// TwinCAT 3 PLC project PI_test
// ProgramVersion: 3.1.4024.0
// libraries:
//   Tc2_ControllerToolbox, * (Beckhoff Automation GmbH)
//   Tc2_Standard, * (Beckhoff Automation GmbH)
//   Tc2_System, * (Beckhoff Automation GmbH)
//   Tc3_Module, * (Beckhoff Automation GmbH)
// project tree:
//   / PlcTask.TcTTO
//   POUs/ FB_FILL_SIM.TcPOU, TYP_VESSEL.TcDUT, MAIN.TcPOU
// real-time tasks:
//   TASK PlcTask: cycle T#1ms, priority 20, ADS port 350

CONFIGURATION PI_test
    RESOURCE PLC ON TwinCAT3
        TASK PlcTask(INTERVAL := T#1ms, PRIORITY := 20);
        PROGRAM MAIN WITH PlcTask : MAIN;
    END_RESOURCE
END_CONFIGURATION

// ---- POUs/TYP_VESSEL.TcDUT
TYPE TYP_VESSEL :
STRUCT
	rVesselSize: LREAL := 100;
	rFillingRate: LREAL := 100;
	rValveInOpening: LREAL := 50;
	rEmptyingRate: LREAL := 100;
	rValveOutOpening: LREAL := 50;
	rSetPoint: LREAL := 50;
	bReset: BOOL;
END_STRUCT
END_TYPE

// ---- POUs/MAIN.TcPOU
PROGRAM MAIN
VAR
	fbVesselSim: FB_FILL_SIM;
	fbPIControl: FB_CTRL_PI;
	stParameters: ST_CTRL_PI_PARAMS;
	gVessel: TYP_VESSEL;
	bChangeDefaultPi: BOOL;
END_VAR

IF NOT bChangeDefaultPi THEN
	stParameters.bARWOnIPartOnly:=FALSE;
	stParameters.fKp:=200; 
	stParameters.fOutMaxLimit:=100; 
	stParameters.fOutMinLimit:=0; 
	stParameters.tCtrlCycleTime:=T#100MS;
	stParameters.tTaskCycleTime:=T#100MS; 
	stParameters.tTn:=T#2M;
END_IF

fbVesselSim(rFillingRate:=gVessel.rFillingRate, 
			rVesselSize:=gVessel.rVesselSize, 
			rValveInOpening:=fbPIControl.fOut, 
			rEmptyingRate:=gVessel.rEmptyingRate, 
			rValveOutOpening:=gVessel.rValveOutOpening, 
			bReset:=gVessel.bReset);

fbPIControl(fSetpointValue:=gVessel.rSetPoint,
			fActualValue:=fbVesselSim.rVesselLevel,
			eMode:=2,
			fManSyncValue := 50,
			bSync:=FALSE,
			bHold:=FALSE,
			stParams:=stParameters);

END_PROGRAM

// ---- POUs/FB_FILL_SIM.TcPOU
FUNCTION_BLOCK FB_FILL_SIM
VAR_INPUT
	rVesselSize: LREAL;
	rFillingRate: LREAL;
	rValveInOpening: LREAL;
	rEmptyingRate: LREAL;
	rValveOutOpening: LREAL;
	bReset: BOOL;
END_VAR
VAR_OUTPUT
	rVesselLevel: LREAL;
	rVesselLevelPercentage: LREAL;
END_VAR
VAR
	rActualFillingRate: LREAL;
	bValveInOpen: BOOL;
	tonTimer1: TON;
	tonTimer2: TON;
	rTrig: R_TRIG;
	bValveOutOpen: BOOL;
	rActualEmptyingRate: LREAL;
END_VAR

bValveInOpen := rValveInOpening > 0;
bValveOutOpen := rValveOutOpening > 0;

rActualFillingRate := rFillingRate*rValveInOpening/100;
rActualEmptyingRate := rEmptyingRate*rValveOutOpening/100;

tonTimer1(IN:=NOT tonTimer2.Q, PT:=T#50MS);
tonTimer2(IN:=tonTimer1.Q, PT:=T#50MS);
rTrig(CLK:=tonTimer1.Q);

IF rTrig.Q THEN
	IF bValveInOpen THEN
		rVesselLevel := rVesselLevel + rActualFillingRate/60000*100;
	END_IF
	IF bValveOutOpen THEN
		rVesselLevel := rVesselLevel - rActualEmptyingRate/60000*100;
	END_IF
END_IF

IF bReset THEN
	rVesselLevel := 0;
END_IF

rVesselLevelPercentage := rVesselLevel/rVesselSize * 100;

END_FUNCTION_BLOCK
